FUNCTION_BLOCK TcCamTable IMPLEMENTS itfCamTable
VAR_INPUT
END_VAR
VAR_OUTPUT
END_VAR
VAR
END_VAR

{warning 'add method implementation '}
METHOD Select 		: itfCommand
VAR_INPUT	
	Periodic		: BOOL;
	MasterAbsolute	: BOOL;
	SlaveAbsolute	: BOOL;
	CamTable		: MC_CAM_REF;
END_VAR
VAR
	
END_VAR
END_METHOD

END_FUNCTION_BLOCK

(* stored: Version 1.1.0.1, ProductVersion 3.1.4024.11
   POU TcCamTable: Id {052b4e8b-1a88-4e87-a422-d46dd3c73661}, SpecialFunc None
   Method Select: Id {02640e26-87dd-44e1-9df6-c10a19b174f6} *)
